//Fifo base control template with external memory based of FifoBase
FUNCTION_BLOCK Fifo EXTENDS FifoBase
VAR_INPUT
END_VAR
VAR_OUTPUT
END_VAR
VAR
END_VAR

;

//Clear out one entry from the Fifo buffer
METHOD PUBLIC clear : BOOL //TRUE if method was successful
VAR_INPUT
	EntryNo													:	UDINT;
	pMemory													: 	POINTER TO BYTE := 0;
	SizeOfMemory											: 	UDINT := 0;
END_VAR             										
VAR                 										
END_VAR
Clear := SUPER^._Clear(EntryNo,pMemory,SizeOfMemory);
END_METHOD

//Clear out defined data set from the Fifo buffer
METHOD PUBLIC clearByDataSet : BOOL //TRUE if method was successful
VAR_INPUT
	pData													: 	POINTER TO BYTE := 0;
	SizeOfData												: 	UDINT := 0;										
	pMemory													: 	POINTER TO BYTE := 0;
	SizeOfMemory											: 	UDINT := 0;
END_VAR             										
VAR         
	i														:	DINT;        										
END_VAR
ClearByDataSet := SUPER^._ClearByDataSet(pData,SizeOfEntry,pMemory,SizeOfMemory);
END_METHOD

METHOD PUBLIC dequeue : BOOL //TRUE if method was successful
VAR_INPUT
	pData													: 	POINTER TO BYTE := 0;
	SizeOfData												: 	UDINT := 0;
	pMemory													: 	POINTER TO BYTE := 0;
	SizeOfMemory											: 	UDINT := 0;
END_VAR
Dequeue := SUPER^._Dequeue(pData,SizeOfEntry,pMemory,SizeOfMemory);
END_METHOD

METHOD PUBLIC enqueue : BOOL //TRUE if method was successful
VAR_INPUT
	pData													: 	POINTER TO BYTE := 0;
	SizeOfData												: 	UDINT := 0;
	pMemory													: 	POINTER TO BYTE := 0;
	SizeOfMemory											: 	UDINT := 0;
END_VAR
Enqueue := SUPER^._Enqueue(pData,SizeOfData,pMemory,SizeOfMemory);
END_METHOD

//Check wheter a value already exist
METHOD PUBLIC isEnqueued : uDINT //data exist in Fifo if reurn value <> 0, returns index of entry in buffer 
VAR_INPUT
	pData													: 	POINTER TO BYTE := 0;
	SizeOfData												: 	UDINT := 0;
	pMemory													: 	POINTER TO BYTE := 0;
	SizeOfMemory											: 	UDINT := 0;
END_VAR	
VAR
	i 														: 	DINT;
END_VAR
IsEnqueued := SUPER^._IsEnqueued(pData,SizeOfEntry,pMemory,SizeOfMemory);
END_METHOD

//Check wheter a value will be the next output of the buffer
METHOD PUBLIC isNextEntry : BOOL //Inputs value is the next output 
VAR_INPUT
	pData													: 	POINTER TO BYTE := 0;
	SizeOfData												: 	UDINT := 0;
	pMemory													: 	POINTER TO BYTE := 0;
	SizeOfMemory											: 	UDINT := 0;
END_VAR
VAR
END_VAR
IsNextEntry := SUPER^._IsNextEntry(pData,SizeOfEntry,pMemory,SizeOfMemory);
END_METHOD

METHOD PUBLIC readEntry : BOOL //TRUE if method was successful
VAR_INPUT
	idx														:	UDINT;
	pData													: 	POINTER TO BYTE := 0;
	SizeOfData												: 	UDINT := 0;
	pMemory													: 	POINTER TO BYTE := 0;
	SizeOfMemory											: 	UDINT := 0;
END_VAR
ReadEntry := SUPER^._ReadEntry(idx,pData,SizeOfEntry,pMemory,SizeOfMemory);
END_METHOD

//Reset complete Fifo
METHOD PUBLIC reset : BOOL //TRUE if method is finnished
VAR_INPUT
	pMemory													: 	POINTER TO BYTE := 0;
	SizeOfMemory											: 	UDINT := 0;
END_VAR
reset := SUPER^._reset(pMemory,SizeOfMemory);
END_METHOD

END_FUNCTION_BLOCK

(* stored: Version 1.1.0.1, ProductVersion 3.1.4024.11
   POU Fifo: Id {aa1f044b-8eab-4938-891f-629e57b9ca73}, SpecialFunc None
   Method clear: Id {fbbef430-ab0a-4417-ad82-366c7bad295c}
   Method clearByDataSet: Id {9fe6205a-3ce0-4f76-90b0-837e52a3b6ee}
   Method dequeue: Id {59de4c4c-74b3-493f-aa4b-ade886aeb471}
   Method enqueue: Id {72027fe0-e175-4e5c-8ae6-cdfc0b7f1938}
   Method isEnqueued: Id {d93336e1-a542-40f1-8838-7b61766d3e75}
   Method isNextEntry: Id {0bc44085-e9b8-4d57-bfa3-96cac1b10e91}
   Method readEntry: Id {75efbd96-7f79-426c-910d-4b1d2a1b3a17}
   Method reset: Id {680644df-fa3c-4296-a961-c8c34a092629} *)
